// TIA Portal V18 export
TYPE "RCS_SysAlarmWarning_V1"
// stored: IsFailsafeCompliant false
   STRUCT
      ON : Bool;   // On Status
      ACK : Bool;   // Acknowledg
      Reset : Bool;
      ImmediatelyStop : Bool;   // Process Immediately Stop
      CycleStop : Bool;   // Process Cycle Stop
   END_STRUCT;
END_TYPE
